TYPE ASCF_CC_OPCUACS_Reader_Interface :
STRUCT
	Connect		: BOOL		:= FALSE;		//Connect the Reader (NOTE: This means the writer will start to read and has nothing to do with the actual OPC UA connection)
	Disconnect	: BOOL		:= FALSE;		//Disconnect the Reader (NOTE: This means the writer will stop to read and has nothing to do with the actual OPC UA connection)
	DoRead		: BOOL		:= FALSE;		//Command to do one read operation. Is set to 0 when done. Use a constant true to continuously read.
	Reset		: BOOL		:= FALSE;		//Reset the Reader
	Config		: ASCF_CC_OPCUACS_ReaderConfig;					//Configuration of the Reader
	Status		: ASCF_CC_OPCUACS_ReaderStatus;					//Status of the Reader
END_STRUCT
END_TYPE

(* stored: Version 1.1.0.1, ProductVersion 3.1.4026.4
   DUT ASCF_CC_OPCUACS_Reader_Interface: Id {93dbbef6-146f-4f9b-be14-8a49658e30d4} *)
